(*
  Table representation of a point
*)
TYPE ST_DeformationPointTbl :
STRUCT
  bSet          : BOOL;
  tTime         : T_DCTIME64;
  sPoint        : ST_DeformationPointAccurate;
END_STRUCT
END_TYPE

(* stored: Version 1.1.0.1, ProductVersion 3.1.4024.11
   DUT ST_DeformationPointTbl: Id {0331c130-84d3-4240-8e8e-57408bf4f9e3} *)
